// TIA Portal V19 export
TYPE "LEXCHANGETRAY_typeSr1000ProfinetTelegram_in"
// stored: Access Published
   STRUCT
      busyStatusBits : "LEXCHANGETRAY_typeSr1000ProfinetTelegram_busyStatusBits";
      completionStatusBits { S7_SetPoint := 'True'} : "LEXCHANGETRAY_typeSr1000ProfinetTelegram_completionStatusBits";
      errorStatusBits { S7_SetPoint := 'True'} : "LEXCHANGETRAY_typeSr1000ProfinetTelegram_errorStatusBits";
      handshakAndGeneralErrorStatusBits { S7_SetPoint := 'True'} : "LEXCHANGETRAY_typeSr1000ProfinetTelegram_handshakAndGeneralErrorStatusBits";
      matchingLevelandTotalEvaluationGradeStatus { S7_SetPoint := 'True'} : "LEXCHANGETRAY_typeSr1000ProfinetTelegram_matchingLevelandTotalEvaluationGradeStatus";
      operationResultStatus { S7_SetPoint := 'True'} : "LEXCHANGETRAY_typeSr1000ProfinetTelegram_operationResultStatus";
      terminalStatusBits { S7_SetPoint := 'True'} : "LEXCHANGETRAY_typeSr1000ProfinetTelegram_terminalStatusBits";
      unstableReadStatusBits { S7_SetPoint := 'True'} : "LEXCHANGETRAY_typeSr1000ProfinetTelegram_unstableReadStatusBits";
      readData128Byte { S7_SetPoint := 'True'} : "LEXCHANGETRAY_typeSr1000ProfinetTelegram_readData128Byte";
   END_STRUCT;
END_TYPE
